TYPE HydraulicsSideProcesses :
STRUCT
	///Reset the drive
	resetDrive: Process;
	///Change the frequency setpoint, in Hertz
	changeFrequencySetpoint: ChangeSetpointProcess;
END_STRUCT
END_TYPE

(* stored: Version 1.1.0.1, ProductVersion 3.1.4019.2
   DUT HydraulicsSideProcesses: Id {90078954-5e0e-4096-a546-1eb2320b7576} *)
